TEXTLIST tlVacuumStep
  1 = 'Init'
  10 = 'Process start'
  15 = 'Waiting for setup pressure'
  20 = 'Waiting for end of cycle'
  25 = 'Cycle ended'
  40 = 'Status change'
  100 = 'Error'
  105 = 'Wait for reset'
  110 = 'Reset in progress'
   = ''
END_TEXTLIST

(* stored: Version 1.1.0.1, ProductVersion 3.1.4024.13
   TextList tlVacuumStep: Id {7d54a0b9-f0b8-4972-87f9-bb16df54d10a} *)
